FUNCTION_BLOCK FB_EuchnerSTP EXTENDS FB_LinkDevice
VAR_INPUT
	bLock 				: BOOL; //Deactivates the tightening magnet
	bLamp_RD			: BOOL; //User defined input for item 1
	bLamp_GN			: BOOL; //User defined input for item 2
END_VAR
VAR_OUTPUT
	bClosed 			: BOOL; //Door is closed
	bClosedAndLocked 	: BOOL; //Door is closed and guard locked / interlocked
END_VAR

SUPER^();
Control.0 			:= bLock;

Control.4 			:= bLamp_RD;
Control.5 			:= bLamp_GN;

bClosed 			:= Status.0;
bClosedAndLocked    := Status.1 OR (bLock AND bClosed);

END_FUNCTION_BLOCK

(* stored: Version 1.1.0.1, ProductVersion 3.1.4024.12
   POU FB_EuchnerSTP: Id {14d65476-a319-058a-356b-e9661403e420}, SpecialFunc None *)
